# EPICS autosave request: iocBoot/ioc1/dbSave/23i_KB_Hy_.req
%
% BURT Request File
%
% 23i:KB:Hy:  Horizontal KB mirror Y-positioning
%

file $(DIR)/assy.req ASSY=23i:KB:Hy
23i:KB:Hy:BaseLength
file $(DIR)/mtr1.req MTR1=23i:KB:mhy1
file $(DIR)/mtr1.req MTR1=23i:KB:mhy2
file $(DIR)/drv1.req DRV1=23i:KB:HY1
file $(DIR)/drv1.req DRV1=23i:KB:HY2
file $(DIR)/axs1.req AXS1=23i:KB:HY
file $(DIR)/axs1.req AXS1=23i:KB:HA
